(* CoDeSys 2.3 export: SENSOR_MAGNETICO.EXP *)

(* Data type *)
TYPE Sensor_Magnetico :
STRUCT
	Activo : BOOL;
END_STRUCT
END_TYPE
